{attribute 'GeneratedUsingTerminal: AT2020-0250-0019'}
{attribute addProperty BoxType "AT2020-0250-0019"}
{attribute addProperty Id "A_0085_AT2050_5500_0018_AT2050_5500AT2050_01D6DEDF80"}
{attribute addProperty CRC "3144771226"}
{attribute addProperty Size "80"}
TYPE A_0060_AT2020_0250_0019_AT2020_0250_BB71669A EXTENDS AT2020_86175B41 :
STRUCT
	{attribute addProperty Name "A_0085_AT2050_5500_0018_AT2050_5500"}
	A_0085_AT2050_5500_0018_AT2050_5500 : AT2050_01D6DEDF;
END_STRUCT
END_TYPE

(* stored: Version 1.2.0.0, ProductVersion 3.1.4024.9
   DUT A_0060_AT2020_0250_0019_AT2020_0250_BB71669A: Id {19794275-527c-450a-9026-143150748ef2} *)
